FUNCTION_BLOCK FB_SQL
VAR_INPUT
END_VAR
VAR_OUTPUT
END_VAR
VAR
	fbSqlDatabase 			:FB_SQLDatabaseEvt(sNetID := '', tTimeout := T#5S);
	fbSqlCommand 			:FB_SQLCommandEvt(sNetID := '', tTimeout := T#5S);
	fbSqlResult 			:FB_SQLResultEvt(sNetID:='', tTimeout := T#5S); 
	fbSQLStoredProcedure	:FB_SQLStoredProcedureEvt(sNetID:='', tTimeout := T#5S);
	
	nStep					:INT;
	nLastStepError			:INT;
	nConnectionStep			:INT;
	
	// Properties
	_Name					:STRING;
	_DBID					:UINT;
	_RecordCounts			:UDINT;
	_Error					:BOOL;
	_ACK					:BOOL;
	_TimeOut				:TIME := T#5S;
END_VAR

IF _Error THEN
	IF nStep <> 200 THEN
		nLastStepError := nStep;
	END_IF
	nStep := 200;
END_IF
IF _Error AND _ACK THEN
	_Error := FALSE;
	nStep := 0;
END_IF
fbSqlDatabase.tTimeout := _TimeOut;
fbSqlCommand.tTimeout := _TimeOut;
fbSqlResult.tTimeout := _TimeOut;
fbSQLStoredProcedure.tTimeout := _TimeOut;

PROPERTY ACK : BOOL
SET
_ACK := ACK;
END_SET
END_PROPERTY

METHOD PRIVATE Connect : BOOL
VAR_INPUT
END_VAR
Connect := FALSE;
IF fbSqlDatabase.bConnected THEN
	Connect := TRUE;
ELSIF fbSqlDatabase.Connect(_DBID) THEN
	IF fbSqlDatabase.bError THEN
		_Error := TRUE;
		Connect := TRUE;
	ELSE
		Connect := TRUE;
	END_IF
END_IF
END_METHOD

METHOD PRIVATE CreateCmd : BOOL
VAR_INPUT
END_VAR
CreateCmd := FALSE;
IF fbSqlDatabase.CreateCmd(ADR(fbSqlCommand)) THEN
	IF fbSqlDatabase.bError THEN
		_Error := TRUE;
		CreateCmd := TRUE;
	ELSE
		CreateCmd := TRUE;
	END_IF
END_IF
END_METHOD

METHOD PRIVATE CreateSP : BOOL
VAR_INPUT
	sProcedureName		:REFERENCE TO STRING;											//Store Procedure name
    pParameterInfo		:POINTER TO ARRAY [0..MAX_SPPARAMETER] OF ST_SQLSPParameter;	//Parameter Info Array
	nParameterInfoSize	:UDINT;															//Size of parameter info array	
END_VAR
CreateSP := FALSE;
IF fbSQLDatabase.CreateSP(sProcedureName, pParameterInfo, nParameterInfoSize, ADR(fbSQLStoredProcedure)) THEN
	IF fbSQLDatabase.bError THEN
		_Error := TRUE;
		CreateSP := TRUE;
	ELSE
		CreateSP := TRUE;
	END_IF
END_IF
END_METHOD

PROPERTY DBID : UINT
GET
DBID := _DBID;
END_GET
END_PROPERTY

METHOD PRIVATE Disconnect : BOOL
VAR_INPUT
END_VAR
Disconnect := FALSE;
IF fbSqlDatabase.Disconnect() THEN
	IF fbSqlDatabase.bError THEN
		_Error := TRUE;
		Disconnect := TRUE;
	ELSE
		nStep := 0;
		Disconnect := TRUE;
	END_IF
END_IF
END_METHOD

PROPERTY Error : BOOL
GET
Error := _Error;
END_GET
END_PROPERTY

METHOD PRIVATE Execute : BOOL
VAR_INPUT
	sCmd		:REFERENCE TO STRING; 	//SQL command
END_VAR
Execute := FALSE;
IF fbSQLCommand.Execute(ADR(sCmd), SIZEOF(sCmd)) THEN
	IF fbSQLCommand.bError THEN
		_Error := TRUE;
		Execute := TRUE;
	ELSE
		Execute := TRUE;  
	END_IF
END_IF
END_METHOD

METHOD PRIVATE ExecuteDataReturn : BOOL
VAR_INPUT
	sCmd		:REFERENCE TO STRING;	//SQL command
END_VAR
ExecuteDataReturn := FALSE;
IF fbSQLCommand.ExecuteDataReturn(ADR(sCmd), SIZEOF(sCmd), ADR(fbSqlResult)) THEN
	IF fbSQLCommand.bError THEN
		_Error := TRUE;
		ExecuteDataReturn := TRUE;
	ELSE
		ExecuteDataReturn := TRUE;
	END_IF
END_IF
END_METHOD

METHOD ExecuteDataReturnSP : BOOL
VAR_INPUT
	pParameterStrc			:POINTER TO BYTE;												//Parameter struct
	nParameterStrcSize		:UDINT;															//Size of parameter struct
END_VAR
ExecuteDataReturnSP := FALSE;
IF fbSQLStoredProcedure.ExecuteDataReturn(pParameterStrc, nParameterStrcSize, ADR(fbSqlResult)) THEN
	IF fbSQLStoredProcedure.bError THEN
		_Error := TRUE;
		ExecuteDataReturnSP := TRUE;
	ELSE
		ExecuteDataReturnSP := TRUE;
	END_IF    
END_IF
END_METHOD

METHOD Init : BOOL
VAR_INPUT
	sName		:REFERENCE TO STRING;
	nDBID		:REFERENCE TO UINT;
	tTimeout	:REFERENCE TO TIME;
END_VAR
_Name := sName;
_DBID := nDBID;
_TimeOut := tTimeout;
Init := TRUE;
END_METHOD

METHOD Modify : BOOL
VAR_INPUT
	sCmd		:REFERENCE TO STRING; 	//SQL command
END_VAR
Modify := FALSE;
CASE nStep OF 
	0:
		IF Connect() THEN
			nStep := nStep + 20; 
		END_IF
	20:
		IF CreateCmd() THEN
			nStep := nStep + 20;  
		END_IF
		
	40:
		IF Execute(sCmd) THEN
			nStep := nStep + 20; 
		END_IF
	
	60: 
		IF Disconnect() THEN
			nStep := 0;
			Modify := TRUE;
		END_IF
		
	200:
		Modify := TRUE;
END_CASE
END_METHOD

PROPERTY Name : STRING
GET
Name := _Name;
END_GET
END_PROPERTY

METHOD PRIVATE Read : BOOL
VAR_INPUT
	pResultRecord			:POINTER TO BYTE;		//Pointer to the struct
	nResultRecordSize		:REFERENCE TO UDINT;	//Size of the struct
END_VAR
Read := FALSE;
_RecordCounts := fbSQLResult.nDataCount;
IF fbSqlResult.Read(0, _RecordCounts, pResultRecord, nResultRecordSize, TRUE, FALSE) THEN
	IF fbSqlResult.bError THEN
		_Error := TRUE;
		Read := TRUE;
	ELSE
		Read := TRUE;
	END_IF
END_IF
END_METHOD

PROPERTY RecordCounts : UDINT
GET
RecordCounts := _RecordCounts;
END_GET
END_PROPERTY

METHOD PRIVATE ReleaseRead : BOOL
VAR_INPUT
END_VAR
ReleaseRead := FALSE;
IF fbSqlResult.Release() THEN
	IF fbSqlResult.bError THEN
		_Error := TRUE;
		ReleaseRead := TRUE;
	ELSE
		ReleaseRead := TRUE; 
	END_IF
END_IF
END_METHOD

METHOD PRIVATE ReleaseSP : BOOL
VAR_INPUT
END_VAR
ReleaseSP := FALSE;
IF fbSQLStoredProcedure.Release() THEN
	IF fbSQLStoredProcedure.bError THEN
		_Error := TRUE;
		ReleaseSP := TRUE;
	ELSE
		ReleaseSP := TRUE;
	END_IF
END_IF
END_METHOD

METHOD Select : BOOL;
VAR_INPUT
	sCmd					:REFERENCE TO STRING;	//SQL command
	pResultRecord			:POINTER TO BYTE;		//Pointer to the struct
	nResultRecordSize		:UDINT;					//Size of the struct
END_VAR
Select := FALSE;
CASE nStep OF 
	0:
		IF Connect() THEN
			nStep := nStep + 20;  
		END_IF
		
	20:
		IF CreateCmd() THEN
			nStep := nStep + 20;  
		END_IF

	40:
		IF ExecuteDataReturn(sCmd) THEN
			nStep := nStep + 20;
		END_IF
		
	60:
		IF Read(pResultRecord, nResultRecordSize) THEN
			nStep := nStep + 20; 
		END_IF
			
	80: 
		IF ReleaseRead() THEN
			nStep := nStep + 20; 
		END_IF
	
	100:
		IF Disconnect() THEN
			nStep := 0;
			Select := TRUE;
		END_IF
		
	200:
		MEMSET(pResultRecord,0, nResultRecordSize);
		_RecordCounts := 0;
		Select := TRUE;
END_CASE
END_METHOD

METHOD StoredProcedure : BOOL
VAR_INPUT
	sProcedureName		:REFERENCE TO STRING;											//Store Procedure name
    pParameterInfo		:POINTER TO ARRAY [0..MAX_SPPARAMETER] OF ST_SQLSPParameter;	//Parameter Info Array
	nParameterInfoSize	:UDINT;															//Size of parameter info array	
	pParameterStrc		:POINTER TO BYTE;												//Parameter struct
	nParameterStrcSize	:UDINT;															//Size of parameter struct
	pResultRecord		:POINTER TO BYTE;												//Pointer to the struct
	nResultRecordSize	:UDINT;															//Size of the struct
END_VAR
StoredProcedure := FALSE;
CASE nStep OF 
	0:
		IF Connect() THEN
			nStep := nStep + 20;  
		END_IF
		
	20:
		IF CreateSP(sProcedureName, pParameterInfo, nParameterInfoSize) THEN
			nStep := nStep + 20;
		END_IF
		
	40:
		IF ExecuteDataReturnSP(pParameterStrc, nParameterStrcSize) THEN
			nStep := nStep + 20;
		END_IF
		
	60:
		IF Read(pResultRecord, nResultRecordSize) THEN
			nStep := nStep + 20; 
		END_IF
			
	80: 
		IF ReleaseRead() THEN
			nStep := nStep + 20; 
		END_IF
		
	100:
		IF ReleaseSP() THEN
			nStep := nStep + 20; 
		END_IF
	
	120:
		IF Disconnect() THEN
			nStep := 0;
			StoredProcedure := TRUE;
		END_IF
		
	200:
		MEMSET(pResultRecord,0, nResultRecordSize);
		_RecordCounts := 0;
		StoredProcedure := TRUE;
END_CASE
END_METHOD

PROPERTY TimeOut : Time
GET
TimeOut := _TimeOut;
END_GET
END_PROPERTY

END_FUNCTION_BLOCK

(* stored: Version 1.1.0.1, ProductVersion 3.1.4024.11
   POU FB_SQL: Id {25a3dc2c-8c6d-41f8-8333-ff0379645580}, SpecialFunc None
   Folder Private_Methods: Id {d634c950-d8ac-49b1-a1be-0fb58c104e98}
   Folder Stored_Procedure: Id {ff1dd28b-212c-4ca4-a8ba-0c01d544df33}
   Folder Properties: Id {3adccdbb-be0a-4a02-a206-4ae9a6d70f6a}
   Property ACK: Id {c627cc4a-1c4b-476e-910c-bcd62be5c497}
   Set Set: Id {cf605164-4724-48c0-93f9-9f721992a384}
   Method Connect: Id {4d302e86-8281-4816-9e97-8d0dec3f2da9}
   Method CreateCmd: Id {42237235-1334-436f-a9c1-ad683f5ea730}
   Method CreateSP: Id {b3b37870-efcb-4472-ba82-a735e985dac7}
   Property DBID: Id {0a98df38-2546-434c-a18c-2e197df4f0bb}
   Get Get: Id {aa6970c6-18be-40d1-aa02-c64c9ae7b917}
   Method Disconnect: Id {0c455447-23db-42fc-827a-ab1e1e45449c}
   Property Error: Id {bc5da951-d167-4c7d-aead-2fabdac99c67}
   Get Get: Id {628ad4d3-0865-4f34-8c58-05c2f984620b}
   Method Execute: Id {55533a9a-bdc0-4dcb-838d-82bde800a588}
   Method ExecuteDataReturn: Id {9b3ed40d-dc04-417b-a9be-3c61b08efc25}
   Method ExecuteDataReturnSP: Id {912d7ff2-26de-40f2-accd-1007bc484aa2}
   Method Init: Id {bea61aaa-73a7-4d4b-8993-e459e9b0248a}
   Method Modify: Id {52defccd-039b-4576-b875-02666d4ef8ca}
   Property Name: Id {094b9ffa-7c7f-4018-a4d3-9688c054cf84}
   Get Get: Id {fe42ac2a-61cd-41fe-80fa-a59f87cccbf4}
   Method Read: Id {a45b5b5e-e55d-4150-a4c4-3eb3f820acf4}
   Property RecordCounts: Id {f61862cf-d449-480b-a2ef-b1e18b210c83}
   Get Get: Id {2d070f0f-9a9c-4b99-a82b-5b9b3692a2fa}
   Method ReleaseRead: Id {c9e4dfed-750c-4f32-affe-9a99df8456cf}
   Method ReleaseSP: Id {8360ab00-3f98-4633-ab92-9c4568929bff}
   Method Select: Id {42cbb836-a9e1-45e7-9618-d7f0136be98f}
   Method StoredProcedure: Id {194d860a-e88c-4885-80ef-8aa2b6fd6f40}
   Property TimeOut: Id {155c609d-3fc8-4018-bf1c-efb02bc8f475}
   Get Get: Id {f233e474-bdce-4f4f-9e26-f243c17b6e8a} *)
